// TIA Portal V20 export
FUNCTION_BLOCK "FB_LoaderFixtureMain"   // FB208, SCL
{ S7_Optimized_Access := 'TRUE' }
// stored: AutoNumber false, MemoryReserve 100, SetENOAutomatically false
   VAR
      sSynchroMode : Bool;
      sSynchroPosition : Bool;
      sTimeMeasure : "FB_TimeMeasure";
      sBlowingNotFinished { S7_SetPoint := 'True'} : Bool;
      sLoadingNotFinished : Bool;
      sUnloadingNotFinished : Bool;
      sReleaseNotFinished : Bool;
      sV_InitNotFinished : Bool;
      sW_InitNotFinished : Bool;
   END_VAR
BEGIN
   REGION Description header 
       //==================================================================================
       // POSALUX Swiss SA / (C) Copyright 2025
       //----------------------------------------------------------------------------------
       // Title: 
       // Comment/Function: 
       // Author: Fabien WALDT
       // Engineering: TIA Portal v17
       //----------------------------------------------------------------------------------
       // Change log table:
       // Version  | Date     | Expert in charge | Changes applied
       // ---------|----------|------------------|-----------------------------------------
       // 00.00.01 | 20251013 | WFA              | First released version
       // =================================================================================
   END_REGION

   REGION Options
       // Fixture
       "DB_LoaderOptions".Fixture.UnloadingDisabled := FALSE;
       "DB_LoaderOptions".Fixture.LoadingDisabled := FALSE;
       "DB_LoaderOptions".Fixture.BlowingDisabled := FALSE;
       "DB_LoaderOptions".Fixture.ReleaseDisabled := TRUE;
       "DB_LoaderOptions".Fixture.V_InitDisabled := FALSE;
       "DB_LoaderOptions".Fixture.W_InitDisabled := FALSE;
   END_REGION

   REGION History Activation
       // Fixture
       "DB_LoaderFixture".sFixtureUnloading.sHistory.Activation := TRUE;
       "DB_LoaderFixture".sFixtureLoading.sHistory.Activation := TRUE;
       "DB_LoaderFixture".sFixtureBlowing.sHistory.Activation := TRUE;
       "DB_LoaderFixture".sFixtureRelease.sHistory.Activation := TRUE;
       "DB_LoaderFixture".sFixtureV_Init.sHistory.Activation := TRUE;
       "DB_LoaderFixture".sFixtureW_Init.sHistory.Activation := TRUE;
   END_REGION

   REGION Fixture
       "DB_LoaderFixture"(iAxisV_Moving:="DB_LoaderAxis".sVPositioning,
                          iAxisV_InPos:="DB_LoaderAxis".sVInPos,
                          iAxisW_Moving:="DB_LoaderAxis".sWPositioning,
                          iAxisW_InPos:="DB_LoaderAxis".sWInPos,
                          oFixtureOpenReq=>"DB_LoaderFixture".oFixtureOpenReq,
                          oFixtureCloseReq=>"DB_LoaderFixture".oFixtureCloseReq,
                          oLoadGripperOpenReq=>"DB_LoaderFixture".oLoadGripperOpenReq,
                          oUnloadGripperCloseReq=>"DB_LoaderFixture".oUnloadGripperCloseReq,
                          oBlowingReq=>"DB_LoaderFixture".oBlowingReq,
                          oAxisV_StartReq=>"DB_LoaderFixture".oAxisV_StartReq,
                          oAxisV_PosSetPoint=>"DB_LoaderFixture".oAxisV_PosSetPoint,
                          oAxisW_StartReq=>"DB_LoaderFixture".oAxisW_StartReq,
                          oAxisW_PosSetPoint=>"DB_LoaderFixture".oAxisW_PosSetPoint);
   END_REGION

   REGION Sequences Not Finished
       IF "DB_LoaderFixture".sFixtureMain.sMemoBlowingRequest THEN
           #sBlowingNotFinished :=
           ("LBP_AlarmMsgs".UserA[08].A70UUxx[11]
           OR "LBP_AlarmMsgs".UserA[08].A70UUxx[10]
           OR "LBP_AlarmMsgs".UserA[08].A70UUxx[12]);
       END_IF;

       IF "DB_LoaderFixture".sFixtureMain.sMemoLoadingRequest THEN
           #sLoadingNotFinished :=
           ("LBP_AlarmMsgs".UserA[08].A70UUxx[11]
           OR "LBP_AlarmMsgs".UserA[08].A70UUxx[10]
           OR "LBP_AlarmMsgs".UserA[08].A70UUxx[12]
           OR "LBP_AlarmMsgs".UserA[08].A70UUxx[14]
           OR "LBP_AlarmMsgs".UserA[08].A70UUxx[13]);
           //  OR "LBP_AlarmMsgs".UserA[04].A70UUxx[26]
       END_IF;

       IF "DB_LoaderFixture".sFixtureMain.sMemoUnloadingRequest THEN
           #sUnloadingNotFinished := 
           ("LBP_AlarmMsgs".UserA[08].A70UUxx[11]
           OR "LBP_AlarmMsgs".UserA[08].A70UUxx[10]
           OR "LBP_AlarmMsgs".UserA[08].A70UUxx[12]
           OR "LBP_AlarmMsgs".UserA[08].A70UUxx[17]);
       END_IF;

       #sReleaseNotFinished := "DB_LoaderFixture".sFixtureRelease.sInterface.SequenceRun AND
       ("LBP_AlarmMsgs".UserA[08].A70UUxx[11]
       OR "LBP_AlarmMsgs".UserA[08].A70UUxx[10]);

       #sV_InitNotFinished := "DB_LoaderFixture".sFixtureV_Init.sInterface.SequenceRun AND
       ("LBP_AlarmMsgs".UserA[08].A70UUxx[10]);

       #sW_InitNotFinished := "DB_LoaderFixture".sFixtureW_Init.sInterface.SequenceRun AND
       ("LBP_AlarmMsgs".UserA[08].A70UUxx[11]);
   END_REGION

   REGION Alarm Not Ready
       // 700515 Gripper not ready for unloading
       IF "DB_LoaderFixture".sFixtureMain.sMemoUnloadingRequest AND NOT "DB_LoaderFixture".sFixtureMain.iGripperReadyForUnloading THEN
           "LBP_AlarmMsgs".UserA[05].A70UUxx[15] := TRUE;
       ELSE
           "LBP_AlarmMsgs".UserA[05].A70UUxx[15] := FALSE;
       END_IF;

       // 700516 Gripper not ready for loading
       IF "DB_LoaderFixture".sFixtureMain.sMemoLoadingRequest AND NOT "DB_LoaderFixture".sFixtureMain.iGripperReadyForLoading THEN
           "LBP_AlarmMsgs".UserA[05].A70UUxx[16] := TRUE;
       ELSE
           "LBP_AlarmMsgs".UserA[05].A70UUxx[16] := FALSE;
       END_IF;

       // 700517 Gripper not ready for blowing
       IF "DB_LoaderFixture".sFixtureMain.sMemoBlowingRequest AND NOT "DB_LoaderFixture".sFixtureMain.iGripperReadyForBlowing THEN
           "LBP_AlarmMsgs".UserA[05].A70UUxx[17] := TRUE;
       ELSE
           "LBP_AlarmMsgs".UserA[05].A70UUxx[17] := FALSE;
       END_IF;

       // 700518 Gripper not ready for V Axis Init
       IF "DB_LoaderFixture".sFixtureMain.sMemoV_InitRequest AND NOT "DB_LoaderFixture".sFixtureMain.iGripperReadyForV_Init THEN
           "LBP_AlarmMsgs".UserA[05].A70UUxx[18] := TRUE;
       ELSE
           "LBP_AlarmMsgs".UserA[05].A70UUxx[18] := FALSE;
       END_IF;

       // 700519 Gripper not ready for W Axis Init 
       IF "DB_LoaderFixture".sFixtureMain.sMemoW_InitRequest AND NOT "DB_LoaderFixture".sFixtureMain.iGripperReadyForW_Init THEN
           "LBP_AlarmMsgs".UserA[05].A70UUxx[19] := TRUE;
       ELSE
           "LBP_AlarmMsgs".UserA[05].A70UUxx[19] := FALSE;
       END_IF;

       // 700520 Fixture not ready for unloading
       IF "DB_LoaderFixture".sFixtureMain.sMemoUnloadingRequest AND NOT "DB_LoaderFixture".sFixtureMain.iFixtureReadyForUnloading THEN
           "LBP_AlarmMsgs".UserA[05].A70UUxx[20] := TRUE;
       ELSE
           "LBP_AlarmMsgs".UserA[05].A70UUxx[20] := FALSE;
       END_IF;

       // 700521 Fixture not ready for loading
       IF "DB_LoaderFixture".sFixtureMain.sMemoLoadingRequest AND NOT "DB_LoaderFixture".sFixtureMain.iFixtureReadyForLoading THEN
           "LBP_AlarmMsgs".UserA[05].A70UUxx[21] := TRUE;
       ELSE
           "LBP_AlarmMsgs".UserA[05].A70UUxx[21] := FALSE;
       END_IF;

       // 700522 Fixture not ready for blowing  
       IF "DB_LoaderFixture".sFixtureMain.sMemoBlowingRequest AND NOT "DB_LoaderFixture".sFixtureMain.iFixtureReadyForBlowing THEN
           "LBP_AlarmMsgs".UserA[05].A70UUxx[22] := TRUE;
       ELSE
           "LBP_AlarmMsgs".UserA[05].A70UUxx[22] := FALSE;
       END_IF;

       // 700523 Fixture not ready for V Axis Init
       IF "DB_LoaderFixture".sFixtureMain.sMemoV_InitRequest AND NOT "DB_LoaderFixture".sFixtureMain.iFixtureReadyForV_Init THEN
           "LBP_AlarmMsgs".UserA[05].A70UUxx[23] := TRUE;
       ELSE
           "LBP_AlarmMsgs".UserA[05].A70UUxx[23] := FALSE;
       END_IF;

       // 700524 Fixture not ready for W Axis Init 
       IF "DB_LoaderFixture".sFixtureMain.sMemoW_InitRequest AND NOT "DB_LoaderFixture".sFixtureMain.iFixtureReadyForW_Init THEN
           "LBP_AlarmMsgs".UserA[05].A70UUxx[24] := TRUE;
       ELSE
           "LBP_AlarmMsgs".UserA[05].A70UUxx[24] := FALSE;
       END_IF;

       // 700525 Axis position not ready for unloading
       IF "DB_LoaderFixture".sFixtureMain.sMemoUnloadingRequest AND NOT "DB_LoaderFixture".sFixtureMain.iAxisReadyForUnloading THEN
           "LBP_AlarmMsgs".UserA[05].A70UUxx[25] := TRUE;
       ELSE
           "LBP_AlarmMsgs".UserA[05].A70UUxx[25] := FALSE;
       END_IF;

       // 700526 Axis position not ready for loading
       IF "DB_LoaderFixture".sFixtureMain.sMemoLoadingRequest AND NOT "DB_LoaderFixture".sFixtureMain.iAxisReadyForLoading THEN
           "LBP_AlarmMsgs".UserA[05].A70UUxx[26] := TRUE;
       ELSE
           "LBP_AlarmMsgs".UserA[05].A70UUxx[26] := FALSE;
       END_IF;

       // 700527 Axis position not ready for blowing
       IF "DB_LoaderFixture".sFixtureMain.sMemoBlowingRequest AND NOT "DB_LoaderFixture".sFixtureMain.iAxisReadyForBlowing THEN
           "LBP_AlarmMsgs".UserA[05].A70UUxx[27] := TRUE;
       ELSE
           "LBP_AlarmMsgs".UserA[05].A70UUxx[27] := FALSE;
       END_IF;

       // 700528 Axis position not ready for V Axis Init
       IF "DB_LoaderFixture".sFixtureMain.sMemoV_InitRequest AND NOT "DB_LoaderFixture".sFixtureMain.iAxisReadyForV_Init THEN
           "LBP_AlarmMsgs".UserA[05].A70UUxx[28] := TRUE;
       ELSE
           "LBP_AlarmMsgs".UserA[05].A70UUxx[28] := FALSE;
       END_IF;

       // 700529 Axis position not ready for W Axis Init 
       IF "DB_LoaderFixture".sFixtureMain.sMemoW_InitRequest AND NOT "DB_LoaderFixture".sFixtureMain.iAxisReadyForW_Init THEN
           "LBP_AlarmMsgs".UserA[05].A70UUxx[29] := TRUE;
       ELSE
           "LBP_AlarmMsgs".UserA[05].A70UUxx[29] := FALSE;
       END_IF;
   END_REGION
END_FUNCTION_BLOCK
